PROGRAM SQLite_CreateDb_V2
VAR_INPUT
	IN_ConfigDbActuelle		: ARRAY[0..MAX_CONFIGURATIONS] OF ST_ConfigDB; 
	IN_DbType				: UINT:= 1; // 1:T_DBConfig_SQLite, 2:T_DBConfig_SQLCe
	IN_Dir					: T_MAXSTRING;
	IN_Name					: STRING;
	IN_Start				: BOOL;
	IN_TableName			: STRING;
END_VAR
VAR_IN_OUT
	IN_hDBID         		: UDINT;	
END_VAR
VAR_OUTPUT
	OUT_Error				: BOOL;
	OUT_Busy				: BOOL;
	OUT_Result				: INT;
END_VAR
VAR
	Etape					: UINT;
	
	TrigStart				: R_TRIG;
	RsStart					: RS;
	bCreateTable			: BOOL;
	TrigCreateTable			: R_TRIG;
	RsCreateTable			: RS;
	PLCDBCreateEvt 			: FB_PLCDBCreateEvt(sNetID := '', tTimeout := T#5S);
	SqlLiteConf				: T_DBConfig_SQLite;
	DbFullDirName			: T_MAXSTRING;	
	sExtension				: STRING:= '.db';
	tcMessage    	 		: I_TcMessage;
	
	AX_ColArray				: ARRAY[0..3] OF ST_ColumnInfo;
	
	dBID_Test				: UDINT;
	KK						: UDINT;
	bExisteDeja				: BOOL;	
END_VAR

OUT_Busy := TRUE;
AX_ColArray[0].sName := 'TimeStamp';     	AX_ColArray[0].eType := E_ColumnType.DateTime;   	AX_ColArray[0].nLength := 4;    
AX_ColArray[1].sName := 'TimeStamp_Ms';    	AX_ColArray[1].eType := E_ColumnType.Integer;    	AX_ColArray[1].nLength := 4;
AX_ColArray[2].sName := 'ParentId';   		AX_ColArray[2].eType := E_ColumnType.Integer;   	AX_ColArray[2].nLength := 4;
AX_ColArray[3].sName := 'Value';   			AX_ColArray[3].eType := E_ColumnType.Float;   		AX_ColArray[3].nLength := 8;


IF IN_DbType = 1 THEN
	sExtension := '.db';
ELSIF IN_DbType = 2 THEN
	sExtension := '.sdf';
END_IF

DbFullDirName := Concat(STR1:=Concat(STR1:= IN_Dir, STR2 := IN_Name), STR2 := sExtension);
SqlLiteConf.bAuthentification := FALSE;
SqlLiteConf.sServer := DbFullDirName;

FOR KK := 0 TO MAX_CONFIGURATIONS DO
	IF IN_ConfigDbActuelle[KK].sServer = DbFullDirName THEN
		bExisteDeja := TRUE;
		OUT_Result := -1;
		OUT_Busy := FALSE;
		OUT_Error := FALSE;
		bCreateTable := FALSE;
		IN_hDBID := IN_ConfigDbActuelle[KK].hDBID;
		EXIT;
	END_IF
	IF KK = MAX_CONFIGURATIONS THEN
		bExisteDeja := FALSE;
	END_IF
END_FOR

TrigStart(CLK := IN_Start AND NOT bExisteDeja);
RsStart(SET := TrigStart.Q);
IF RsStart.Q1 THEN
	IF PLCDBCreateEvt.Database(pDatabaseConfig := ADR(SqlLiteConf), cbDatabaseConfig := SIZEOF(SqlLiteConf), bCreateXMLConfig := TRUE, pDBID := ADR(dBID_Test)) THEN
		IF PLCDBCreateEvt.ipTcResult.nEventId = 59 THEN
			OUT_Error := FALSE;
			OUT_Result := -1;
			OUT_Busy := FALSE;	
			TrigStart(CLK := FALSE);
			bCreateTable := FALSE;
			Etape := 0;
			RsCreateTable(RESET1 := TRUE);
			RsCreateTable(RESET1 := FALSE);
		ELSIF PLCDBCreateEvt.bError THEN
			tcMessage := PLCDBCreateEvt.ipTcResult;
			OUT_Error := TRUE;
		ELSE
			Etape := 1;
			IN_hDBID := dBID_Test;
			bCreateTable := TRUE; 
		END_IF
		RsStart(RESET1 := TRUE);
		RsStart(RESET1 := FALSE);
	END_IF
END_IF

TrigCreateTable(CLK := bCreateTable);
RsCreateTable(SET:= TrigCreateTable.Q);

IF RsCreateTable.Q1 AND ETAPE = 1 THEN
	IF PLCDBCreateEvt.Table(hDBID := IN_hDBID, sTableName := IN_TableName,  pTableCfg := ADR(AX_ColArray), cbTableCfg := SIZEOF(AX_ColArray)  ) THEN
		IF PLCDBCreateEvt.bError THEN
			Etape := 255;
			OUT_Error := TRUE;
			OUT_Result := -2;
		ELSE
			IN_Start := FALSE;
			bCreateTable := FALSE;
			Etape := 0;
			OUT_Result := 1;
			RsCreateTable(RESET1 := TRUE);
			RsCreateTable(RESET1 := FALSE);
			TrigStart(CLK := False);
			OUT_Busy := FALSE;	
			OUT_Error := FALSE;
		END_IF
	END_IF
END_IF

IF Etape = 255 THEN
	Etape := 0;
	bCreateTable := FALSE;
	IN_Start := FALSE;
	OUT_Busy := FALSE;	
	RsCreateTable(RESET1 := TRUE);
	RsCreateTable(RESET1 := FALSE);
	
END_IF

END_PROGRAM

(* stored: Version 1.1.0.1, ProductVersion 3.1.4024.6
   POU SQLite_CreateDb_V2: Id {dd2eff89-efd6-40f9-95eb-d095892ada03}, SpecialFunc None *)
